TYPE ST_ECYCtrl :
STRUCT
    bServON   :BOOL;   
    bHome      :BOOL;   
    bReset      :BOOL;   
    bStop         :BOOL;   
   bJog_P         :BOOL;   
   bJog_N        :BOOL;   
   Pos_Start      :BOOL;   
   fTagetPos     :REAL;
   fVel:           REAL;
   fAcc        :REAL;  
   fDec        :REAL;  
  // Delay_Time  :TIME;


     bHomed         :BOOL; 
     Pos_Done       :BOOL;   //定位完成
     Home_Alm      :BOOL;  //回零超时报警
     Pos_Alm         :BOOL; //定位超时报警



END_STRUCT
END_TYPE

(* stored: Version 1.1.0.1, ProductVersion 3.1.4024.9
   DUT ST_ECYCtrl: Id {34c5c8ed-994b-47c3-b111-8fec4344f76f} *)
